// Mitsubishi GX Works2 project: k06   PLC: Q02/Q02H

PROGRAM MAIN
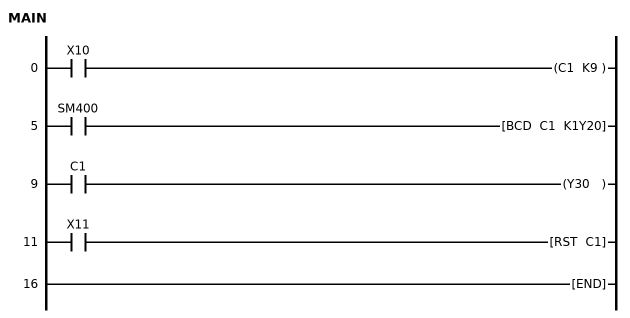
0     LD      X10
      OUT     C1 K9
5     LD      SM400
      BCD     C1 K1Y20
9     LD      C1
      OUT     Y30
11    LD      X11
      RST     C1
16    END
END_PROGRAM
